PROGRAM MAIN
VAR
	increment 			: BOOL;
	counter 			: INT;
	
	incrementTrigger	: R_TRIG;		
END_VAR

incrementTrigger(CLK := increment);

IF incrementTrigger.Q THEN
	counter := (counter + 1) MOD 11;
END_IF

END_PROGRAM

(* stored: Version 1.1.0.1, ProductVersion 3.1.4024.13
   POU MAIN: Id {8a9825f3-734c-4350-ad0b-60f99cb3afcb}, SpecialFunc None *)
